	E_MA_EVENT.STOP_TRACK:
		RefStat.sm.sEventDesc := 'CMD STOP_TRACK';
		RETURN;
		
	E_MA_EVENT.PRESETDONE:
		RefStat.sm.sEventDesc := 'TRACKING';
		RETURN;
		
	E_MA_EVENT.TRACKEXIT:
		RefStat.sm.sEventDesc := 'TRACKING -> PRESETTING';
		RETURN;
		
	E_MA_EVENT.HWOK:
		RefStat.sm.sEventDesc := 'SIG HWOK';
		RETURN;

	E_MA_EVENT.ERRHW:
		RefStat.sm.sEventDesc := 'INT ERRHW';
		RETURN;
	
END_CASE 

(* INTERNAL ERROR *)
RefStat.sm.sEventDesc := 'UNKNOWN EVENT';
END_METHOD

// Set the state and substate of the device
METHOD SetState : BOOL
VAR_INPUT
	in_nState:		INT;
	in_nSubstate:	INT;
END_VAR

(* 
	Update State Machine active state configuration.
*)

IF in_nState <> E_MA_STATE.NONE THEN
	RefStat.sm.nState	:= in_nState;
END_IF
IF in_nSubstate <> E_MA_SUBSTATE.NONE THEN
	RefStat.sm.nSubstate	:= in_nSubstate;
END_IF

(* Update active state configuration description *)

IF in_nState = E_MA_STATE.NOTOP THEN
	RefStat.sm.sState	:= 'NOT OP';
ELSIF in_nState = E_MA_STATE.OP THEN
	RefStat.sm.sState	:= 'OPERATIONAL';
END_IF

IF in_nSubstate = E_MA_SUBSTATE.NOTOP_NOTREADY THEN
	RefStat.sm.sSubstate	:= 'NOT READY';
ELSIF in_nSubstate = E_MA_SUBSTATE.NOTOP_INITIALISING THEN
	RefStat.sm.sSubstate	:= 'INITIALISING';
ELSIF in_nSubstate = E_MA_SUBSTATE.NOTOP_READY THEN
	RefStat.sm.sSubstate	:= 'READY';
ELSIF in_nSubstate = E_MA_SUBSTATE.NOTOP_ERROR THEN
	RefStat.sm.sSubstate	:= 'ERROR';
ELSIF in_nSubstate = E_MA_SUBSTATE.OP_DISABLING THEN
	RefStat.sm.sSubstate	:= 'DISABLING';
ELSIF in_nSubstate = E_MA_SUBSTATE.OP_MOVING THEN
	RefStat.sm.sSubstate	:= 'MOVING';
ELSIF in_nSubstate = E_MA_SUBSTATE.OP_STANDSTILL THEN
	RefStat.sm.sSubstate	:= 'STANDSTILL';
ELSIF in_nSubstate = E_MA_SUBSTATE.OP_TRACKING THEN
	RefStat.sm.sSubstate	:= 'TRACKING';
ELSIF in_nSubstate = E_MA_SUBSTATE.OP_PRESETTING THEN
	RefStat.sm.sSubstate	:= 'PRESETTING';
ELSIF in_nSubstate = E_MA_SUBSTATE.OP_STOPPING THEN
	RefStat.sm.sSubstate	:= 'STOPPING';
ELSIF in_nSubstate = E_MA_SUBSTATE.OP_ERROR THEN
	RefStat.sm.sSubstate	:= 'ERROR';
ELSE
	RefStat.sm.sSubstate	:= '';
END_IF
END_METHOD

METHOD User_ComputeNextPos : BOOL
VAR_INPUT
END_VAR
VAR
	i:	int;
END_VAR
// TODOUSER: Calculate next position for each axes based on the current mode.
IF RefStat.nMode = MA_MODE_ENG THEN
	FOR i := 1 TO nNumAxes DO
		;
	END_FOR
END_IF
END_METHOD

// Method for hard-coding of configuration parameters by the User.
METHOD User_Configure : BOOL
VAR_INPUT
END_VAR
VAR
	i:	INT;
END_VAR
//
// TODOUSER: Configure anything that is different from default configuration or
//           that has to take all motors into account.
//

//
// This is mandatory.
//
// Set the global timeouts to the longest ones. 
FOR i := 1 TO nNumAxes DO
	IF ptrMotorCfg[i]^.nTimeoutInit > RefCfg.tout.initTime THEN
		RefCfg.tout.initTime  := ptrMotorCfg[i]^.nTimeoutInit;
	END_IF
	IF ptrMotorCfg[i]^.nTimeoutMove > RefCfg.tout.moveTime THEN
		RefCfg.tout.moveTime  := ptrMotorCfg[i]^.nTimeoutMove;
	END_IF
END_FOR

//
// TODOUSER: Any other configuration
//
END_METHOD

// User Method executed on each cycle before processing events and states.
METHOD User_GetParams : BOOL
VAR_INPUT
END_VAR
VAR
	i:	INT;
END_VAR
//
// TODOUSER: Set anything that should be set on every cycle, if any.
//

// Example: Any settings that are mode dependant.
CASE RefCtrl.nMode OF
			MA_MODE_ENG:
			    ; 
END_CASE
END_METHOD

// User Method executed on each cycle after processing events and states.
METHOD User_SetParams : BOOL
VAR_INPUT
END_VAR
VAR
	i:		INT;
END_VAR
//
// Mandatory
//
// Set maximum positioning error
RefStat.lrPosError	:= M_GetMaxPosError();


// TODO Add code for handling individual axes, if any.
FOR i := 1 TO nNumAxes DO
	;
END_FOR
END_METHOD

END_FUNCTION_BLOCK

// POUs/MultiAxis/FB_MA_DROT
FUNCTION_BLOCK FB_MA_DROT EXTENDS FB_TRK_BASE
VAR_INPUT
	{attribute 'OPC.UA.DA' := '0'}
	sMotorName:			STRING	:= 'Motor';	(* Default Motor name *)
	{attribute 'OPC.UA.DA' := '0'}
	nNOVRAM_DevId:	UDINT	:= 0;		(* NOVRAM device ID - normally 4 *)
	{attribute 'OPC.UA.DA' := '0'}
	nNOVRAM_Offset:	UDINT	:= 0;		(* NOVRAM offset where motor configuration is stored *)
END_VAR
VAR_OUTPUT
END_VAR
VAR

	
	{attribute 'OPC.UA.DA' := '1'}
	cfg:				T_DROT_CFG;
	{attribute 'OPC.UA.DA' := '1'}
	ctrl:				T_DROT_CTRL;
	{attribute 'OPC.UA.DA' := '1'}
	stat:				T_DROT_STAT;
	
	{attribute 'OPC.UA.DA':='1'}
	motor:              FB_MOTOR;
	
END_VAR


// A MUST !!! Set references to real structures
RefCfg		REF=cfg;
RefCtrl		REF=ctrl;
RefStat		REF=stat;
TrkStat		REF=stat;
TrkCfg      REF=cfg;
TrkCtrl     REF=ctrl;

motor(sName := sMotorName,	nNOVRAM_DevId := nNOVRAM_DevId, nNOVRAM_Offset := nNOVRAM_Offset);
SUPER^(nNumAxes:=1, pMotor1:=ADR(motor));

METHOD M_LogCommand : BOOL
VAR
	cmd:	INT;
	mode:	int;
END_VAR
cmd		:= RefCtrl.nCommand;
mode	:= ctrl.nMode;

// Log DROT command.
// Set motor logging to FALSE when tracking,
// in order to reduce flooding of logs.
IF cmd = E_MA_COMMAND.RESET THEN
	pMotor1^.RPC_SetLog(TRUE);
	M_SetStatus('Resetting DROT device...');		
	M_LogEventGeneral('Resetting DROT device...');
ELSIF cmd = E_MA_COMMAND.ENABLE THEN
	pMotor1^.RPC_SetLog(TRUE);
	M_SetStatus('');		
	M_LogEventGeneral('Enabling DROT device...');
ELSIF cmd = E_MA_COMMAND.INIT THEN
	pMotor1^.RPC_SetLog(TRUE);
	M_SetStatus('Initialising DROT device...');		
	M_LogEventGeneral('Initialising DROT device...');
ELSIF cmd = E_MA_COMMAND.START_TRACK THEN
	pMotor1^.RPC_SetLog(FALSE);
	IF mode= E_DROT_MODE.ELEV THEN
		M_SetStatus('Tracking in ELEV mode');
		M_LogEventGeneral('Setting DROT device to ELEVATION mode...');
	ELSIF mode= E_DROT_MODE.SKY THEN
		M_SetStatus('Tracking in SKY mode');
		M_LogEventGeneral('Setting DROT device to SKY mode...');
	ELSIF mode= E_DROT_MODE.USER THEN
		M_SetStatus('Tracking in USER mode');
		M_LogEventGeneral('Setting DROT device to USER mode...');
	END_IF
ELSIF cmd = E_MA_COMMAND.DISABLE THEN
	M_SetStatus('');		
	M_LogEventGeneral('Disabling DROT device...');
ELSIF cmd = E_MA_COMMAND.STOP THEN
	pMotor1^.RPC_SetLog(TRUE);
	M_LogEventGeneral('Stopping DROT device...');
ELSIF cmd = E_MA_COMMAND.STOP_TRACK THEN
	pMotor1^.RPC_SetLog(TRUE);
	IF mode= E_DROT_MODE.ENG THEN
		M_SetStatus('Moving to Engineering position ...');		
		M_LogEventGeneral('Setting DROT device to ENGINEERING mode...');
	ELSIF mode= E_DROT_MODE.STAT THEN
		M_SetStatus('Moving to STAT position ...');		
		M_LogEventGeneral('Setting DROT device to STAT mode...');
	END_IF
END_IF
END_METHOD

{attribute 'TcRpcEnable':='1'}
METHOD RPC_Disable : INT
VAR_INPUT
END_VAR

// It does all the verifications for the MOTOR device before
// triggering the Init event.

// RPC calls are not allowed in Local mode.
IF ptrMotorStat[1]^.bLocal THEN
	RPC_Disable	:= M_SetRpcStatus(E_MA_RPC_ERROR.LOCAL);
	RETURN;
END_IF

// Disable command is accepted only if device is in OP state.
IF ptrMotorStat[1]^.nState <> E_MOTOR_STATE.OP THEN
	RPC_Disable	:= M_SetRpcStatus(E_MA_RPC_ERROR.NOT_OP);
	RETURN;
ELSE
	// Set disable command
	RefCtrl.nCommand := E_MA_COMMAND.DISABLE;
	RefCtrl.bExecute := TRUE;
	
	// Call was successful
	RPC_Disable	:= M_SetRpcStatus(E_MA_RPC_ERROR.OK);
END_IF
END_METHOD

{attribute 'TcRpcEnable':='1'}
METHOD RPC_Enable : INT
VAR_INPUT
END_VAR

// It does all the verifications for the MOTOR device before
// triggering the Init event.


// RPC calls are not allowed in Local mode.
IF ptrMotorStat[1]^.bLocal THEN
	RPC_Enable	:= M_SetRpcStatus(E_MA_RPC_ERROR.LOCAL);
	RETURN;
END_IF

// Enable command is accepted only if device is in NOTOP_READY.
IF	ptrMotorStat[1]^.nSubstate <> E_MOTOR_SUBSTATE.NOTOP_READY		THEN
	RPC_Enable	:= M_SetRpcStatus(E_MA_RPC_ERROR.NOT_NOTOP_READY);
	RETURN;
ELSE
	// Set enable command
	RefCtrl.nCommand := E_MA_COMMAND.ENABLE;
	RefCtrl.bExecute := TRUE;
	
	// Call was successful
	RPC_Enable	:= M_SetRpcStatus(E_MA_RPC_ERROR.OK);
END_IF
END_METHOD

{attribute 'TcRpcEnable':='1'}
METHOD RPC_Init : INT
VAR_INPUT
END_VAR

VAR
END_VAR
M_LogEventGeneral('Initialising DROT motor...');

RPC_Init	:= SUPER^.RPC_Init();
END_METHOD

{attribute 'TcRpcEnable':='1'}
METHOD RPC_MoveAbs : INT
VAR_INPUT
	in_lrPos:	LREAL;
	in_lrVel:	LREAL;
END_VAR
// RPC calls are not allowed in Local mode.
IF motor.stat.bLocal THEN
	RPC_MoveAbs	:= M_SetRpcStatus(E_MA_RPC_ERROR.LOCAL);
	RETURN;
// Move Absolute command is accepted only in OP state.
ELSIF	motor.stat.nState <> E_MOTOR_STATE.OP	THEN
	RPC_MoveAbs	:= M_SetRpcStatus(E_MA_RPC_ERROR.NOT_OP);
	RETURN;
ELSIF	stat.sm.nState <> E_MA_STATE.OP	THEN
	RPC_MoveAbs	:= M_SetRpcStatus(E_MA_RPC_ERROR.NOT_OP);
	RETURN;
// Set velocity cannot be <=0.0.
ELSIF	in_lrVel <= 0.0	THEN
	RPC_MoveAbs	:= M_SetRpcStatus(E_MOTOR_RPC_ERROR.VEL_NEG);
	RETURN;
// Set velocity cannot be greater than MAX Velocity.
ELSIF	in_lrVel > motor.stat.axis.lrMaxVelocity	THEN
	RPC_MoveAbs	:= M_SetRpcStatus(E_MOTOR_RPC_ERROR.VEL_MAX);
	RETURN;
END_IF


SetState(E_MA_STATE.OP, E_MA_SUBSTATE.OP_MOVING);
// Set command
ctrl.nCommand 		:= E_MA_COMMAND.MA_MOVE;
ctrl.nMode          := E_DROT_MODE.ENG;
ctrl.lrTargetPos    := in_lrPos;
ctrl.lrTargetVel    := in_lrVel;
ctrl.bExecute 		:= TRUE;

// Call was successful
RPC_MoveAbs	:= M_SetRpcStatus(E_MA_RPC_ERROR.OK);
END_METHOD

{attribute 'TcRpcEnable':='1'}
METHOD RPC_MoveAngle : INT
VAR_INPUT
	in_lrAngle:	LREAL;
END_VAR

// RPC calls are not allowed in Local mode.
IF motor.stat.bLocal THEN
	RPC_MoveAngle	:= M_SetRpcStatus(E_MA_RPC_ERROR.LOCAL);
	RETURN;
// Move Absolute command is accepted only in OP state.
ELSIF	motor.stat.nState <> E_MOTOR_STATE.OP	THEN
	RPC_MoveAngle	:= M_SetRpcStatus(E_MA_RPC_ERROR.NOT_OP);
	RETURN;
ELSIF	stat.sm.nState <> E_MA_STATE.OP	THEN
	RPC_MoveAngle	:= M_SetRpcStatus(E_MA_RPC_ERROR.NOT_OP);
	RETURN;
END_IF


SetState(E_MA_STATE.OP, E_MA_SUBSTATE.OP_MOVING);
// Set command
ctrl.lrPosang 	:= in_lrAngle;
ctrl.nMode		:= E_DROT_MODE.STAT;
ctrl.nCommand	:= E_MA_COMMAND.STOP_TRACK;
ctrl.bExecute	:= TRUE;

// Call was successful
RPC_MoveAngle	:= M_SetRpcStatus(E_MA_RPC_ERROR.OK);
END_METHOD

{attribute 'TcRpcEnable':='1'}
METHOD RPC_MoveRel : INT
VAR_INPUT
	in_lrPos:	LREAL;
	in_lrVel:	LREAL;
END_VAR
// RPC calls are not allowed in Local mode.
IF motor.stat.bLocal THEN
	RPC_MoveRel	:= M_SetRpcStatus(E_MA_RPC_ERROR.LOCAL);
	RETURN;
// Move Absolute command is accepted only in OP state.
ELSIF	motor.stat.nState <> E_MOTOR_STATE.OP	THEN
	RPC_MoveRel	:= M_SetRpcStatus(E_MA_RPC_ERROR.NOT_OP);
	RETURN;
ELSIF	stat.sm.nState <> E_MA_STATE.OP	THEN
	RPC_MoveRel	:= M_SetRpcStatus(E_MA_RPC_ERROR.NOT_OP);
	RETURN;
// Set velocity cannot be <=0.0.
ELSIF	in_lrVel <= 0.0	THEN
	RPC_MoveRel	:= M_SetRpcStatus(E_MOTOR_RPC_ERROR.VEL_NEG);
	RETURN;
// Set velocity cannot be greater than MAX Velocity.
ELSIF	in_lrVel > motor.stat.axis.lrMaxVelocity	THEN
	RPC_MoveRel	:= M_SetRpcStatus(E_MOTOR_RPC_ERROR.VEL_MAX);
	RETURN;
END_IF


SetState(E_MA_STATE.OP, E_MA_SUBSTATE.OP_MOVING);
// Set command
ctrl.nCommand 		:= E_MA_COMMAND.MA_MOVE;
ctrl.nMode          := E_DROT_MODE.ENG;
ctrl.lrTargetPos    := motor.stat.lrPosActual + in_lrPos;
ctrl.lrTargetVel    := in_lrVel;
ctrl.bExecute 		:= TRUE;

// Call was successful
RPC_MoveRel	:= M_SetRpcStatus(E_MA_RPC_ERROR.OK);
END_METHOD

{attribute 'TcRpcEnable':='1'}
METHOD RPC_MoveVel : INT
VAR_INPUT
	in_lrVel:	LREAL;
END_VAR
VAR
	dir:	DINT;
END_VAR
IF	stat.sm.nState <> E_MA_STATE.OP	THEN
	RPC_MoveVel	:= M_SetRpcStatus(E_MA_RPC_ERROR.NOT_OP);
	RETURN;
ELSIF	in_lrVel = 0.0	THEN
// Set velocity cannot be 0.0.
	RPC_MoveVel	:= M_SetRpcStatus(E_MOTOR_RPC_ERROR.VEL_ZERO);
	RETURN;
END_IF

// Check velocity against Vel_max.
// Note: Negative velocity is accepted.
// Check if Velocity is too high.
IF ABS(in_lrVel) > ptrMotorStat[1]^.axis.lrMaxVelocity THEN
	RPC_MoveVel	:= M_SetRpcStatus(E_MOTOR_RPC_ERROR.VEL_MAX);
	RETURN;
END_IF


// Update State and Status
SetState(E_MA_STATE.OP, E_MA_SUBSTATE.OP_MOVING);
M_SetStatus('Moving in Velocity mode...');
ctrl.nMode	:= E_ADC_MODE.ENG;

// Set the direction of movement.
IF in_lrVel > 0.0	THEN
	dir	:= MC_Positive_Direction;
ELSE
	dir	:= MC_Negative_Direction;
END_IF

// This will command all the motors and restart the timer.
ActionMoveVelExecute(vel:=ABS(in_lrVel), dir:=dir);

// Call was successful
RPC_MoveVel	:= M_SetRpcStatus(E_MA_RPC_ERROR.OK);
END_METHOD

{attribute 'TcRpcEnable':='1'}
METHOD RPC_Reset : INT
VAR_INPUT
END_VAR

// RPC calls are not allowed in Local mode.
IF ptrMotorStat[1]^.bLocal THEN
	RPC_Reset	:= M_SetRpcStatus(E_MA_RPC_ERROR.LOCAL);
	RETURN;
END_IF

ctrl.nCommand := E_MA_COMMAND.RESET;
ctrl.bExecute := TRUE;

// Call was successful
RPC_Reset	:= M_SetRpcStatus(E_MA_RPC_ERROR.OK);
END_METHOD

{attribute 'TcRpcEnable':='1'}
METHOD RPC_StartTrack : INT
VAR_INPUT
	in_mode:	 INT := 2;
	in_angle:    LREAL := 0.0;
END_VAR

// RPC calls are not allowed in Local mode.
IF ptrMotorStat[1]^.bLocal THEN
	RPC_StartTrack	:= M_SetRpcStatus(E_MA_RPC_ERROR.LOCAL);
	RETURN;
// Move Absolute command is accepted only in OP state.
ELSIF	ptrMotorStat[1]^.nState <> E_MOTOR_STATE.OP	THEN
	RPC_StartTrack	:= M_SetRpcStatus(E_MA_RPC_ERROR.NOT_OP);
	RETURN;
END_IF

// Set command
ctrl.lrPosang := in_angle;
ctrl.nMode:= in_mode;
ctrl.nCommand:=E_MA_COMMAND.START_TRACK;
ctrl.bExecute:=(TRUE);

// Call was successful
RPC_StartTrack	:= M_SetRpcStatus(E_MA_RPC_ERROR.OK);
END_METHOD

{attribute 'TcRpcEnable':='1'}
METHOD RPC_Stop : INT
VAR_INPUT
END_VAR

// RPC calls are not allowed in Local mode.
IF ptrMotorStat[1]^.bLocal THEN
	RPC_Stop	:= M_SetRpcStatus(E_MA_RPC_ERROR.LOCAL);
	RETURN;
END_IF

ctrl.nCommand := E_MA_COMMAND.STOP;
ctrl.bExecute := TRUE;

RPC_Stop	:= M_SetRpcStatus(E_MA_RPC_ERROR.OK);
END_METHOD

{attribute 'TcRpcEnable':='1'}
METHOD RPC_StopTrack : INT
VAR_INPUT
END_VAR

IF (RefStat.nMode >= E_DROT_MODE.SKY) THEN
	// RPC calls are not allowed in Local mode.
	IF ptrMotorStat[1]^.bLocal THEN
		RPC_StopTrack	:= M_SetRpcStatus(E_MA_RPC_ERROR.LOCAL);
		RETURN;
	END_IF

	RefCtrl.nMode           :=  E_DROT_MODE.STAT;
	// Set command
	RefCtrl.nCommand 		:= E_MA_COMMAND.STOP_TRACK;
	RefCtrl.bExecute 		:= TRUE;
END_IF

// Call was successful
RPC_StopTrack	:= M_SetRpcStatus(E_MA_RPC_ERROR.OK);
END_METHOD

METHOD User_ComputeNextPos : BOOL
VAR_INPUT
END_VAR
VAR
	fieldRotation: LREAL;
	modeAngle:     LREAL;
	pos:           LREAL := 0.0 ;
	posang:        LREAL;
END_VAR
// Handle various derotator modes
CASE RefCtrl.nMode OF
			E_DROT_MODE.STAT:
			    pos := cfg.lrStatRef + cfg.nDirSign * (ctrl.lrPosang)/2.0;
				stat.lrAngleOnSky := 0.0;
				stat.lrModeAngle := pos;
				ptrMotorCtrl[1]^.lrVelocity := ptrMotorCfg[1]^.lrDefaultVelocity;
			E_DROT_MODE.SKY:
				fieldRotation := stat.data.pa_deg - cfg.nFocusSign * stat.data.alt_deg;
				pos := cfg.lrSkyRef + cfg.nDirSign * (ctrl.lrPosang - fieldRotation)/2;
				stat.lrAngleOnSky := ctrl.lrPosang;
				stat.lrModeAngle := stat.lrAngleOnSky;
				ptrMotorCtrl[1]^.lrVelocity := ptrMotorCfg[1]^.lrDefaultVelocity;
			E_DROT_MODE.ELEV:
				pos := cfg.lrElevRef + (cfg.nFocusSign * cfg.nDirSign * stat.data.alt_deg) /2.0;
				stat.lrAngleOnSky := stat.data.pa_deg;
				stat.lrModeAngle := stat.lrAngleOnSky;
				ptrMotorCtrl[1]^.lrVelocity := ptrMotorCfg[1]^.lrDefaultVelocity;
			E_DROT_MODE.USER:
				//modeAngle := (parUser[1] * ctrl.lrPosang +
				//	          parUser[2] * i_trk_data.alt_deg +
				//			  parUser[3] * i_trk_data.pa_deg );
				//pos := cfg.lrUserRef + cfg.nDirSign * modeAngle;
				//stat.lrAngleOnSky := 0.0;
				//stat.lrModeAngle  := modeAngle;
			E_DROT_MODE.ENG:
				pos := ctrl.lrTargetPos;
		        ptrMotorCtrl[1]^.lrVelocity := ctrl.lrTargetVel;		
		        M_SetStatus('Moving to Engineering position ...');
END_CASE

// assign new TARGET position
ptrMotorCtrl[1]^.lrPosition := pos;
stat.lrPos := pos;	// Used in the DROT GUI as 'Target'
END_METHOD

// Method for hard-coding of configuration parameters by the User.
METHOD User_Configure : BOOL
VAR_INPUT
END_VAR
VAR
	i:	INT;
END_VAR
SUPER^.User_Configure();	// Mandatory!

//
// TODOUSER: Configure anything that is different from default configuration.
//
// Examples:
//

//
// Individual Motor configuration
ptrMotorCfg[1]^.nAxisType	        := E_MOTOR_AXIS_TYPE.CIRCULAR_OPTIMISED;
ptrMotorCfg[1]^.lrDefaultVelocity	:= 3.0;	// Set default velocity to 10 deg/sec


// Multi-axis system configuration
ctrl.lrPosang	    :=  0.0;	// Position angle for OFF mode, i.e. HOME position
ctrl.lrTargetPos	:=  0.0;	
ctrl.lrTargetVel	:= 3.0;	// Velocity for ENG mode
END_METHOD

// User Method executed on each cycle before processing events and states.
METHOD User_GetParams : BOOL
VAR_INPUT
END_VAR
VAR
	i:	INT;
END_VAR


SUPER^.User_GetParams();
END_METHOD

// User Method executed on each cycle after processing events and states.
METHOD User_SetParams : BOOL
VAR_INPUT
END_VAR
VAR
	i:		INT;
END_VAR
//
// Mandatory
//
SUPER^.User_SetParams();

// Set maximum positioning error
stat.lrPosError		:= M_GetMaxPosError();

// Check if we are tracking or still presetting.
// Tracking is OK if the positioning error is less than the threshold (bTrackingOK).
// Once device is tracking, it should go back to presetting if the error is greater
// than twice the threshold  (bTrackingBAD).
IF	ctrl.nMode = E_DROT_MODE.ELEV OR  
	ctrl.nMode = E_DROT_MODE.SKY  OR  
	ctrl.nMode = E_DROT_MODE.USER	THEN
	stat.bTrackingOK	:= SEL (stat.lrPosError <= cfg.lrTrkThreshold, FALSE, TRUE);
	stat.bTrackingBAD	:= SEL (stat.lrPosError > 2.0 * cfg.lrTrkThreshold, FALSE, TRUE);
ELSE
	stat.bTrackingOK	:= FALSE;
	stat.bTrackingBAD	:= FALSE;
END_IF
END_METHOD

END_FUNCTION_BLOCK

// VISUs/Motor/GUI_Motor001_Cfg
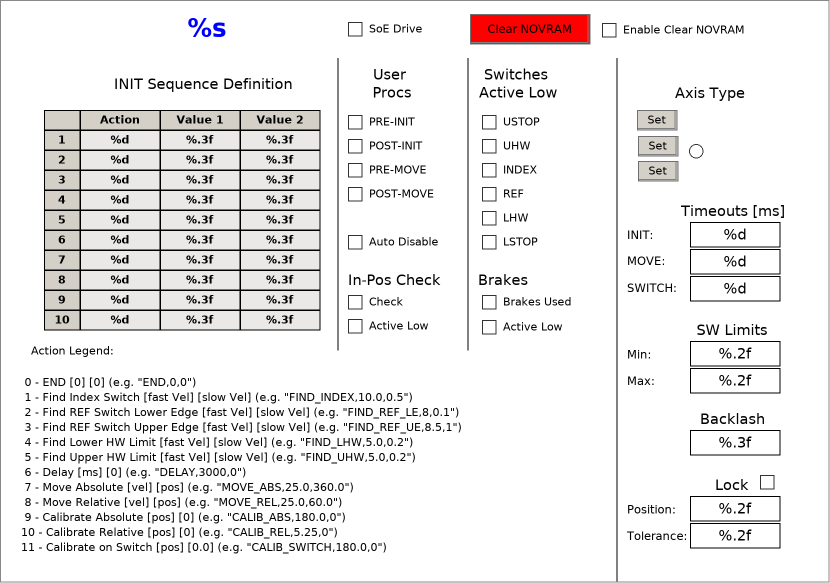
VISUALIZATION GUI_Motor001_Cfg  // 830x583
    Frame (0,0 828x581)
        shows GUI_TEMPLATE_MOTOR_CONFIG(m_Instance := MAIN.Motor001)
END_VISUALIZATION

// VISUs/Motor/GUI_Motor001_Ctrl
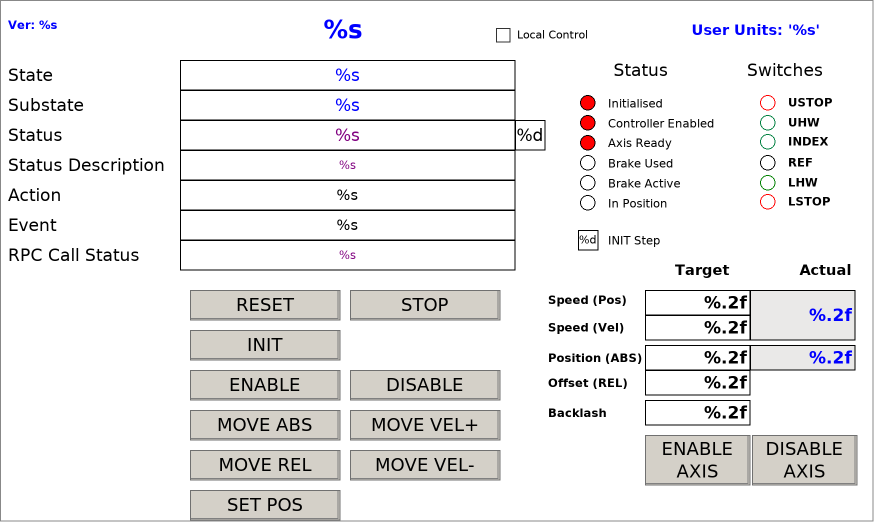
VISUALIZATION GUI_Motor001_Ctrl  // 874x522
    Frame (0,0 872x520)
        shows GUI_TEMPLATE_MOTOR_CONTROL(m_Instance := MAIN.Motor001)
END_VISUALIZATION

// VISUs/Motor/GUI_Motor002_Cfg
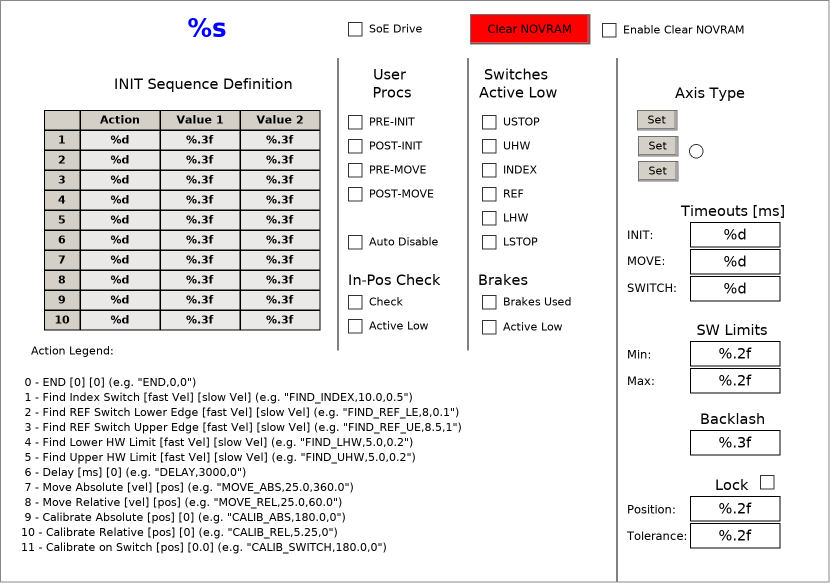
VISUALIZATION GUI_Motor002_Cfg  // 830x583
    Frame (0,0 828x581)
        shows GUI_TEMPLATE_MOTOR_CONFIG(m_Instance := MAIN.Motor002)
END_VISUALIZATION

// VISUs/Motor/GUI_Motor002_Ctrl
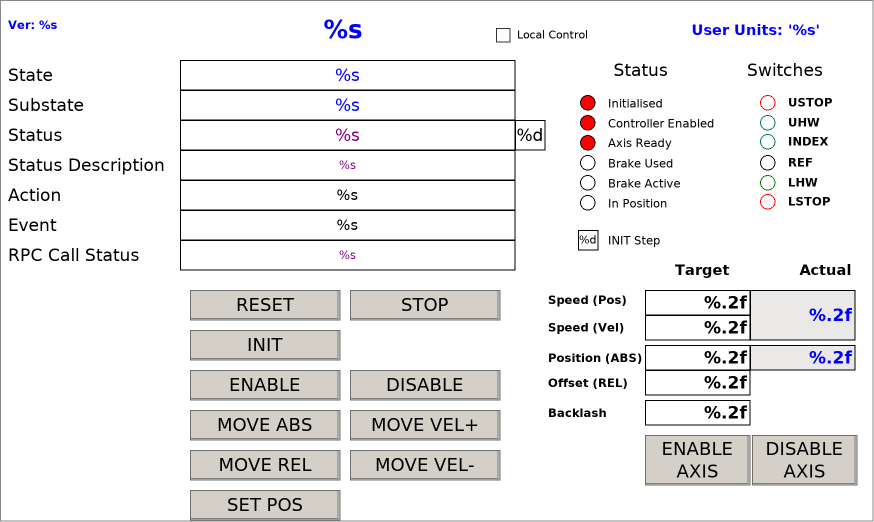
VISUALIZATION GUI_Motor002_Ctrl  // 874x522
    Frame (0,0 872x520)
        shows GUI_TEMPLATE_MOTOR_CONTROL(m_Instance := MAIN.Motor002)
END_VISUALIZATION

// VISUs/Templates/GUI_TEMPLATE_CCS_SIM
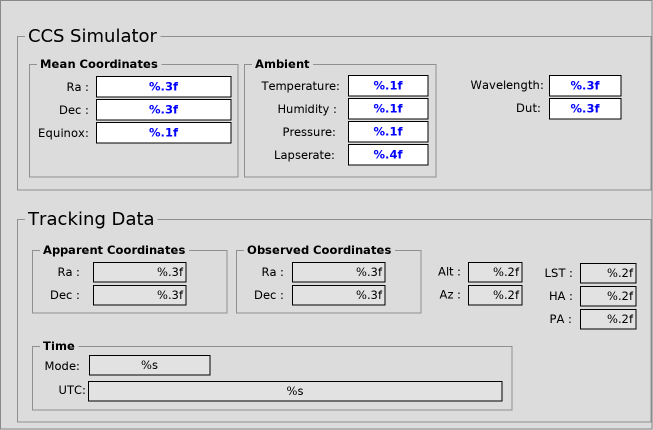
VISUALIZATION GUI_TEMPLATE_CCS_SIM  // 653x430
VAR_INPUT
	m_DeviceName : STRING;
END_VAR
VAR_IN_OUT
	m_Instance : FB_CCS_SIM;
END_VAR
    GroupBox (17,28 634x162), "CCS Simulator"
        GroupBox (12,28 209x121), "Mean Coordinates"
            Label (23,21 40x20), "Ra :"
            Label (23,44 40x20), "Dec :"
            Rectangle (67,20 135x21), "%.3f", tooltip "Mean Right Ascension [hhmmss]", text variable: m_Instance.ctrl.meanCoordinates.alpha
                OnMouseDown: write the text variable via Edit
            Rectangle (67,43 135x21), "%.3f", tooltip "Mean Declination [ddmmss]", text variable: m_Instance.ctrl.meanCoordinates.delta
                OnMouseDown: write the text variable via Edit
            Rectangle (67,66 135x21), "%.1f", tooltip "Equinox", text variable: m_Instance.ctrl.meanCoordinates.equinox
                OnMouseDown: write the text variable via Edit
            Label (3,67 60x20), "Equinox:"
        GroupBox (227,28 192x121), "Ambient"
            Label (7,20 92x20), "Temperature:"
            Label (17,43 79x20), "Humidity :"
            Rectangle (104,19 80x21), "%.1f", tooltip "Temperature [degC]", text variable: m_Instance.ctrl.environment.temperature
                OnMouseDown: write the text variable via Edit
            Rectangle (104,42 80x21), "%.1f", tooltip "Humidity [%]", text variable: m_Instance.ctrl.environment.humidity
                OnMouseDown: write the text variable via Edit
            Rectangle (104,65 80x21), "%.1f", tooltip "Pressure [mbar]", text variable: m_Instance.ctrl.environment.pressure
                OnMouseDown: write the text variable via Edit
            Label (25,66 70x20), "Pressure:"
            Label (24,89 70x20), "Lapserate:"
            Rectangle (104,88 80x21), "%.4f", tooltip "Lapse Rate", text variable: m_Instance.ctrl.environment.lapserate
                OnMouseDown: write the text variable via Edit
        Rectangle (532,47 72x21), "%.3f", text variable: m_Instance.ctrl.wavelength
            OnMouseDown: write the text variable via Edit
        Rectangle (532,70 72x21), "%.3f", text variable: m_Instance.ctrl.dut
            OnMouseDown: write the text variable via Edit
        Label (481,70 46x20), "Dut:"
    GroupBox (17,211 634x211), "Tracking Data"
        GroupBox (15,31 195x71), "Apparent Coordinates"
            Label (11,20 40x20), "Ra :"
            Label (11,43 40x20), "Dec :"
            Label (8,70 60x20)
            Rectangle (61,43 93x20), "%.3f", tooltip "Apparent Declination [ddmmss]", text variable: m_Instance.stat.apparent.delta
            Rectangle (61,20 93x20), "%.3f", tooltip "Apparent Right Ascension [hhmmss]", text variable: m_Instance.stat.apparent.alpha
        Rectangle (563,98 56x20), "%.2f", tooltip "Parallactic Angle [deg]", text variable: m_Instance.stat.data.pa_deg
        Label (508,98 50x20), "PA :"
        Label (410,51 37x19), "Alt :"
        Label (412,74 35x19), "Az :"
        GroupBox (219,31 185x71), "Observed Coordinates"
            Label (11,20 40x20), "Ra :"
            Label (11,43 40x20), "Dec :"
            Label (8,70 60x20)
            Rectangle (56,20 93x20), "%.3f", tooltip "Observed Right Ascension [hhmmss]", text variable: m_Instance.stat.observed.alpha
            Rectangle (56,43 93x20), "%.3f", tooltip "Observed Declination [ddmmss]", text variable: m_Instance.stat.observed.delta
        Rectangle (451,74 54x20), "%.2f", tooltip "TEL Azimuth [deg]", text variable: m_Instance.stat.data.az_deg
        Rectangle (451,51 54x20), "%.2f", tooltip "TEL Altitude [deg]", text variable: m_Instance.stat.data.alt_deg
        GroupBox (15,127 480x72), "Time"
            Label (11,18 40x20), "Mode:"
            Label (11,42 46x20), "UTC:"
            Label (8,70 60x20)
            Rectangle (57,17 121x20), "%s", tooltip "Time mode [UTC, Local or Simulation]", text variable: m_Instance.stat.sTimeMode
            Rectangle (56,43 414x20), "%s", tooltip "Actual time", text variable: m_Instance.stat.sDcTime
    Label (464,75 83x20), "Wavelength:"
    Label (526,263 50x20), "LST :"
    Label (526,286 50x20), "HA :"
    Rectangle (580,286 56x20), "%.2f", tooltip "Hour Angle [deg]", text variable: m_Instance.stat.data.ha
    Rectangle (580,263 56x20), "%.2f", tooltip "Local Sidereal Time [h]", text variable: m_Instance.stat.data.lst
END_VISUALIZATION

// VISUs/Templates/GUI_TEMPLATE_MA_ADC
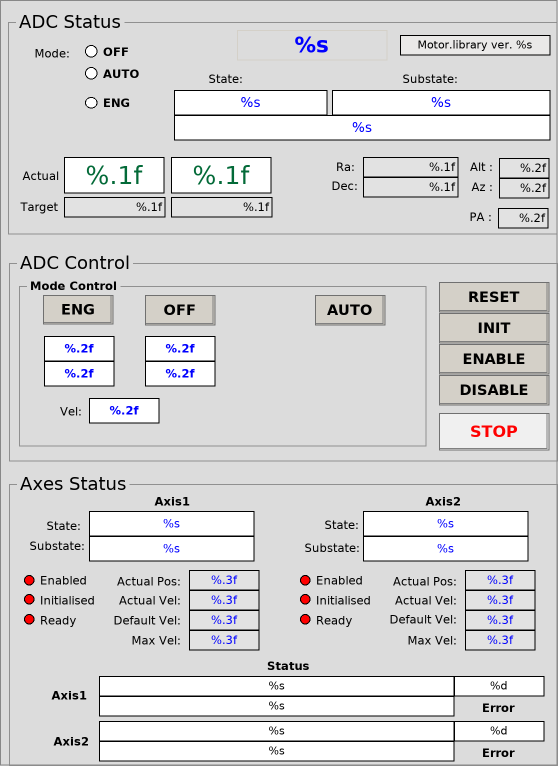
VISUALIZATION GUI_TEMPLATE_MA_ADC  // 558x766
VAR_INPUT
	m_DeviceName : STRING;
END_VAR
VAR_IN_OUT
	m_Instance : FB_MA_ADC;
END_VAR
    GroupBox (9,255 549x206), "ADC Control"
        Button (430,158 110x37), "STOP"
            OnMouseClick: execute { m_Instance.ctrl.nCommand:= E_MA_COMMAND.STOP; m_Instance.ctrl.bExecute:=(TRUE); }
        GroupBox (10,23 407x168), "Mode Control"
            Button (296,17 70x30), "AUTO", tooltip "Tracking mode (2)"
                OnMouseClick: execute {
                    m_Instance.ctrl.nMode:= E_ADC_MODE.AUTO;
                    m_Instance.ctrl.nCommand:=E_MA_COMMAND.START_TRACK;
                    m_Instance.ctrl.bExecute:=(TRUE);
                }
            Rectangle (70,120 70x25), "%.2f", tooltip "Velocity for Engineering Mode [deg/sec]", text variable: m_Instance.ctrl.lrTargetVel
                OnMouseDown: write the text variable via Edit
            Button (126,17 70x30), "OFF", tooltip "OFF (HOME) mode (1)"
                OnMouseClick: execute {
                    m_Instance.ctrl.nMode:=E_ADC_MODE.OFF;
                    m_Instance.ctrl.nCommand:= E_MA_COMMAND.STOP_TRACK;
                    m_Instance.ctrl.bExecute:=(TRUE);
                }
            Label (36,121 30x25), "Vel:"
            Rectangle (126,58 70x25), "%.2f", tooltip "ADC1 OFF Position angle [deg]", text variable: m_Instance.ctrl.lrPosang[1]
                OnMouseDown: write the text variable via Edit
            Rectangle (126,83 70x25), "%.2f", tooltip "ADC2 OFF position angle [deg]", text variable: m_Instance.ctrl.lrPosang[2]
                OnMouseDown: write the text variable via Edit
            Button (24,17 70x29), "ENG", tooltip "ENG mode (0)"
                OnMouseClick: execute {
                    m_Instance.ctrl.nMode:=E_ADC_MODE.ENG;
                    m_Instance.ctrl.nCommand:= E_MA_COMMAND.STOP_TRACK;
                    m_Instance.ctrl.bExecute:=(TRUE);
                }
            Rectangle (25,58 70x25), "%.2f", tooltip "ADC1 ENG Position angle [deg]", text variable: m_Instance.ctrl.lrTargetPos[1]
                OnMouseDown: write the text variable via Edit
        Button (430,120 110x30), "DISABLE"
            OnMouseClick: execute { m_Instance.ctrl.nCommand:= E_MA_COMMAND.DISABLE; m_Instance.ctrl.bExecute:=(TRUE); }
        Button (430,27 110x30), "RESET"
            OnMouseClick: execute { m_Instance.ctrl.nCommand:= E_MA_COMMAND.RESET; m_Instance.ctrl.bExecute:=(TRUE); }
        Button (430,89 110x30), "ENABLE"
            OnMouseClick: execute { m_Instance.ctrl.nCommand:= E_MA_COMMAND.ENABLE; m_Instance.ctrl.bExecute:=(TRUE); }
        Button (430,58 110x30), "INIT"
            OnMouseClick: execute { m_Instance.ctrl.nCommand:= E_MA_COMMAND.INIT; m_Instance.ctrl.bExecute:=(TRUE); }
    GroupBox (9,476 549x290), "Axes Status"
        Label (98,93 77x25), "Actual Pos:"
        Rectangle (180,94 70x20), "%.3f", tooltip "[deg]", text variable: m_Instance.pMotor1^.stat.lrPosActual
        Rectangle (180,114 70x20), "%.3f", tooltip "[deg/sec]", text variable: m_Instance.pMotor1^.stat.lrVelActual
        Label (28,117 70x15), "Initialised"
        Label (28,97 70x15), "Enabled"
        Ellipse (15,118 10x10), tooltip "GREEN=Initialised RED=NOT Initialised", colour toggle: (m_Instance.pMotor1^.stat.bInitialised) <> 0
        Label (105,112 70x25), "Actual Vel:"
        Label (227,180 105x20), "Status"
        Label (437,222 105x20), "Error"
        Rectangle (90,220 355x20), "%s", tooltip "Error Description", text variable: m_Instance.pMotor1^.stat.sErrorText
        Label (28,137 70x15), "Ready"
        Ellipse (15,138 10x10), tooltip "GREEN=Initialised RED=NOT Initialised", colour toggle: (m_Instance.pMotor1^.stat.bAxisReady) <> 0
        Rectangle (90,200 355x20), "%s", tooltip "Motor Status", text variable: m_Instance.pMotor1^.stat.sStatus
        Rectangle (445,200 90x20), "%d", tooltip "Error ID", text variable: m_Instance.pMotor1^.stat.nErrorCode
        Label (94,132 81x25), "Default Vel:"
        Rectangle (180,134 70x20), "%.3f", tooltip "[deg/sec]", text variable: m_Instance.pMotor1^.cfg.lrDefaultVelocity
        Rectangle (80,35 165x25), "%s", text variable: m_Instance.pMotor1^.stat.sState
        Label (12,55 67x30), "Substate:"
        Rectangle (90,245 355x20), "%s", tooltip "Motor Status", text variable: m_Instance.pMotor2^.stat.sStatus
        Label (29,35 46x30), "State:"
        Label (437,267 105x20), "Error"
        Rectangle (354,35 165x25), "%s", text variable: m_Instance.pMotor2^.stat.sState
        Rectangle (80,60 165x25), "%s", text variable: m_Instance.pMotor1^.stat.sSubstate
        Rectangle (354,60 165x25), "%s", text variable: m_Instance.pMotor2^.stat.sSubstate
        Label (287,57 67x30), "Substate:"
        Label (308,34 45x30), "State:"
        Label (136,13 55x25), "Axis1"
        Label (408,13 53x25), "Axis2"
        Label (26,207 55x25), "Axis1"
        Ellipse (15,99 10x10), tooltip "GREEN=Enabled RED=NOT Enabled", colour toggle: (m_Instance.pMotor1^.stat.bEnabled) <> 0
        Ellipse (291,118 10x10), tooltip "GREEN=Initialised RED=NOT Initialised", colour toggle: (m_Instance.pMotor2^.stat.bInitialised) <> 0
        Label (105,152 70x25), "Max Vel:"
        Label (381,152 70x25), "Max Vel:"
    GroupBox (8,14 549x220), "ADC Status"
        Label (10,26 69x27), "Mode:"
        Ellipse (77,83 12x11), tooltip "Engineering Mode: WHITE=Not active GREEN=Activated", colour toggle: (m_Instance.stat.nMode) = E_ADC_MODE.ENG
        Ellipse (77,31 12x12), tooltip "Stationary Mode: WHITE=Not Active GREEN=Activated", colour toggle: (m_Instance.stat.nMode) = E_ADC_MODE.OFF
        Label (92,80 35x18), "ENG"
        Ellipse (77,53 12x12), tooltip "Sky Mode: WHITE=Not Active GREEN=Activated", colour toggle: (m_Instance.stat.nMode) = E_ADC_MODE.AUTO
        Label (92,28 90x20), "OFF"
        Label (310,143 40x20), "Ra:"
        Label (313,162 40x20), "Dec:"
        Rectangle (355,143 95x20), "%.1f", tooltip "TEL RA", text variable: m_Instance.stat.apparent.alpha
        Rectangle (355,163 95x20), "%.1f", tooltip "TEL Dec", text variable: m_Instance.stat.apparent.delta
        Rectangle (490,194 50x20), "%.2f", tooltip "Parallactic Angle [deg]", text variable: m_Instance.stat.data.pa_deg
        Label (437,193 50x20), "PA :"
        Rectangle (491,144 50x20), "%.2f", tooltip "TEL Altitude [deg]", text variable: m_Instance.stat.data.alt_deg
        Rectangle (491,164 50x20), "%.2f", tooltip "TEL Azimuth [deg]", text variable: m_Instance.stat.data.az_deg
        Label (438,143 50x20), "Alt :"
        Label (438,163 50x20), "Az :"
        Rectangle (324,76 218x25), "%s", text variable: m_Instance.stat.sm.sSubstate
        Rectangle (166,76 153x25), "%s", text variable: m_Instance.stat.sm.sState
        Rectangle (166,101 376x25), "%s", text variable: m_Instance.stat.sStatus
        Label (193,50 45x30), "State:"
        Rectangle (392,21 150x20), "Motor.library ver. %s", text variable: m_Instance.stat.sLibVersion
        Rectangle (229,16 150x30), "%s", text variable: m_DeviceName
        Label (389,50 64x30), "Substate:"
        Rectangle (56,143 100x36), "%.1f", text variable: m_Instance.pMotor1^.stat.lrPosActual
        Label (6,179 47x28), "Target"
        Rectangle (56,183 101x20), "%.1f", tooltip "Motor 1 target position in user units (UU).", text variable: m_Instance.pMotor1^.stat.lrPosTarget
        Label (7,148 47x28), "Actual"
        Label (92,50 45x20), "AUTO"
        Rectangle (163,143 100x36), "%.1f", text variable: m_Instance.pMotor2^.stat.lrPosActual
        Rectangle (163,183 101x20), "%.1f", tooltip "Motor 2 target position in user units (UU).", text variable: m_Instance.pMotor2^.stat.lrPosTarget
    Label (447,721 105x20), "Error"
    Rectangle (99,741 355x20), "%s", tooltip "Error Description", text variable: m_Instance.pMotor2^.stat.sErrorText
    Label (37,729 55x25), "Axis2"
    Rectangle (454,721 90x20), "%d", tooltip "Error ID", text variable: m_Instance.pMotor2^.stat.nErrorCode
    Label (382,569 78x25), "Actual Pos:"
    Rectangle (465,570 70x20), "%.3f", tooltip "[deg]", text variable: m_Instance.pMotor2^.stat.lrPosActual
    Rectangle (465,590 70x20), "%.3f", tooltip "[deg/sec]", text variable: m_Instance.pMotor2^.stat.lrVelActual
    Label (313,593 70x15), "Initialised"
    Label (313,573 70x15), "Enabled"
    Label (390,588 70x25), "Actual Vel:"
    Label (313,613 70x15), "Ready"
    Label (377,607 83x25), "Default Vel:"
    Rectangle (465,610 70x20), "%.3f", tooltip "[deg/sec]", text variable: m_Instance.pMotor2^.cfg.lrDefaultVelocity
    Ellipse (300,614 10x10), tooltip "GREEN=Initialised RED=NOT Initialised", colour toggle: (m_Instance.pMotor2^.stat.bAxisReady) <> 0
    Ellipse (300,575 10x10), tooltip "GREEN=Enabled RED=NOT Enabled", colour toggle: (m_Instance.pMotor2^.stat.bEnabled) <> 0
    Rectangle (44,361 70x25), "%.2f", tooltip "ADC2 ENG position angle [deg]", text variable: m_Instance.ctrl.lrTargetPos[2]
        OnMouseDown: write the text variable via Edit
    Rectangle (189,630 70x20), "%.3f", tooltip "[deg/sec]", text variable: m_Instance.pMotor1^.stat.axis.lrMaxVelocity
    Rectangle (465,630 70x20), "%.3f", tooltip "[deg/sec]", text variable: m_Instance.pMotor2^.stat.axis.lrMaxVelocity
END_VISUALIZATION

// VISUs/Templates/GUI_TEMPLATE_MA_DROT
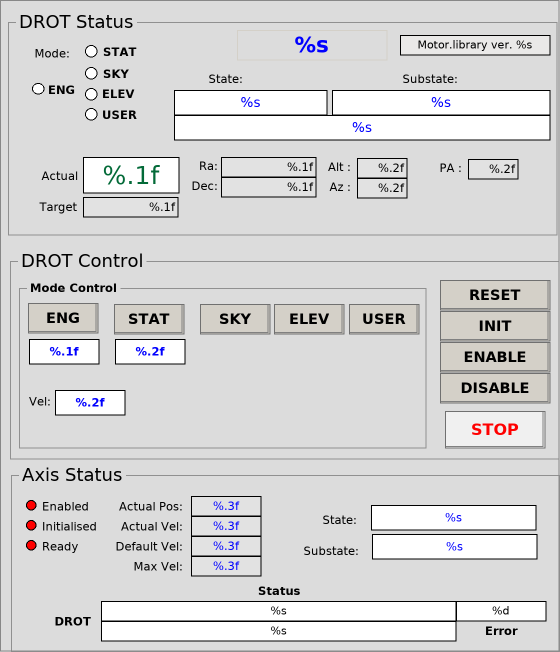
VISUALIZATION GUI_TEMPLATE_MA_DROT  // 560x652
VAR_INPUT
	m_DeviceName : STRING;
END_VAR
VAR_IN_OUT
	m_Instance : FB_MA_DROT;
END_VAR
    GroupBox (10,253 549x206), "DROT Control"
        Button (435,158 100x37), "STOP"
            OnMouseClick: execute { m_Instance.ctrl.nCommand:= E_MA_COMMAND.STOP; m_Instance.ctrl.bExecute:=(TRUE); }
        GroupBox (9,27 407x168), "Mode Control"
            Button (181,24 70x30), "SKY", tooltip "SKY mode (2)"
                OnMouseClick: execute {
                    m_Instance.ctrl.nMode:= E_DROT_MODE.SKY;
                    m_Instance.ctrl.nCommand:=E_MA_COMMAND.START_TRACK;
                    m_Instance.ctrl.bExecute:=(TRUE);
                }
            Rectangle (10,59 70x25), "%.1f", tooltip "[deg]", text variable: m_Instance.ctrl.lrTargetPos
                OnMouseDown: write the text variable via Edit
            Button (9,23 70x30), "ENG", tooltip "Engineering mode (0)"
                OnMouseClick: execute {
                    m_Instance.ctrl.nMode:= E_DROT_MODE.ENG;
                    m_Instance.ctrl.nCommand:= E_MA_COMMAND.STOP_TRACK;
                    m_Instance.ctrl.bExecute:=(TRUE);
                }
            Rectangle (36,110 70x25), "%.2f", tooltip "Velocity for Engineering Mode [deg/sec]", text variable: m_Instance.ctrl.lrTargetVel
                OnMouseDown: write the text variable via Edit
            Button (255,24 70x30), "ELEV", tooltip "ELEV mode (3)"
                OnMouseClick: execute {
                    m_Instance.ctrl.nMode:= E_DROT_MODE.ELEV;
                    m_Instance.ctrl.nCommand:=E_MA_COMMAND.START_TRACK;
                    m_Instance.ctrl.bExecute:=(TRUE);
                }
            Button (95,24 70x30), "STAT", tooltip "STAT mode (1)"
                OnMouseClick: execute {
                    m_Instance.ctrl.nMode:=E_DROT_MODE.STAT;
                    m_Instance.ctrl.nCommand:= E_MA_COMMAND.STOP_TRACK;
                    m_Instance.ctrl.bExecute:=(TRUE);
                }
            Button (330,24 70x30), "USER", tooltip "USER mode (4)"
                OnMouseClick: execute {
                    m_Instance.ctrl.nMode:= E_DROT_MODE.USER;
                    m_Instance.ctrl.nCommand:=E_MA_COMMAND.START_TRACK;
                    m_Instance.ctrl.bExecute:=(TRUE);
                }
            Label (5,109 30x25), "Vel:"
            Rectangle (96,59 70x25), "%.2f", tooltip "Position angle [deg]", text variable: m_Instance.ctrl.lrPosang
                OnMouseDown: write the text variable via Edit
        Button (430,120 110x30), "DISABLE"
            OnMouseClick: execute { m_Instance.ctrl.nCommand:= E_MA_COMMAND.DISABLE; m_Instance.ctrl.bExecute:=(TRUE); }
        Button (430,27 110x30), "RESET"
            OnMouseClick: execute { m_Instance.ctrl.nCommand:= E_MA_COMMAND.RESET; m_Instance.ctrl.bExecute:=(TRUE); }
        Button (430,89 110x30), "ENABLE"
            OnMouseClick: execute { m_Instance.ctrl.nCommand:= E_MA_COMMAND.ENABLE; m_Instance.ctrl.bExecute:=(TRUE); }
        Button (430,58 110x30), "INIT"
            OnMouseClick: execute { m_Instance.ctrl.nCommand:= E_MA_COMMAND.INIT; m_Instance.ctrl.bExecute:=(TRUE); }
    GroupBox (11,467 549x185), "Axis Status"
        Label (105,27 70x25), "Actual Pos:"
        Rectangle (180,29 70x20), "%.3f", tooltip "[deg]", text variable: m_Instance.pMotor1^.stat.lrPosActual
        Rectangle (180,49 70x20), "%.3f", tooltip "[deg/sec]", text variable: m_Instance.pMotor1^.stat.lrVelActual
        Label (28,52 70x15), "Initialised"
        Ellipse (15,33 10x10), tooltip "GREEN=Enabled RED=NOT Enabled", colour toggle: (m_Instance.pMotor1^.stat.bEnabled) <> 0
        Label (28,32 70x15), "Enabled"
        Ellipse (15,53 10x10), tooltip "GREEN=Initialised RED=NOT Initialised", colour toggle: (m_Instance.pMotor1^.stat.bInitialised) <> 0
        Label (105,47 70x25), "Actual Vel:"
        Label (216,114 105x20), "Status"
        Label (438,154 105x20), "Error"
        Rectangle (90,154 355x20), "%s", tooltip "Error Description", text variable: m_Instance.pMotor1^.stat.sErrorText
        Label (28,142 55x25), "DROT"
        Label (28,72 70x15), "Ready"
        Ellipse (15,73 10x10), tooltip "GREEN=Initialised RED=NOT Initialised", colour toggle: (m_Instance.pMotor1^.stat.bAxisReady) <> 0
        Rectangle (90,134 355x20), "%s", tooltip "Motor Status", text variable: m_Instance.pMotor1^.stat.sStatus
        Rectangle (445,134 90x20), "%d", tooltip "Error ID", text variable: m_Instance.pMotor1^.stat.nErrorCode
        Label (105,67 70x25), "Default Vel:"
        Rectangle (180,69 70x20), "%.3f", tooltip "[deg/sec]", text variable: m_Instance.pMotor1^.cfg.lrDefaultVelocity
        Rectangle (360,38 165x25), "%s", text variable: m_Instance.pMotor1^.stat.sState
        Label (259,38 90x30), "State:"
        Label (261,69 90x30), "Substate:"
        Rectangle (361,67 165x25), "%s", text variable: m_Instance.pMotor1^.stat.sSubstate
        Label (105,87 70x25), "Max Vel:"
        Rectangle (180,89 70x20), "%.3f", tooltip "[deg/sec]", text variable: m_Instance.pMotor1^.stat.axis.lrMaxVelocity
    GroupBox (8,14 549x221), "DROT Status"
        Label (10,26 69x27), "Mode:"
        Ellipse (24,69 12x11), tooltip "Engineering Mode: WHITE=Not active GREEN=Activated", colour toggle: (m_Instance.stat.nMode) = E_DROT_MODE.ENG
        Ellipse (77,31 12x12), tooltip "Stationary Mode: WHITE=Not Active GREEN=Activated", colour toggle: (m_Instance.stat.nMode) = E_DROT_MODE.STAT
        Label (37,67 83x18), "ENG"
        Ellipse (77,53 12x12), tooltip "Sky Mode: WHITE=Not Active GREEN=Activated", colour toggle: (m_Instance.stat.nMode) = E_DROT_MODE.SKY
        Ellipse (77,74 12x12), tooltip "Elevation Mode: WHITE=Not Active GREEN=Activated", colour toggle: (m_Instance.stat.nMode) = E_DROT_MODE.ELEV
        Label (91,70 43x20), "ELEV"
        Label (92,50 45x20), "SKY"
        Label (92,28 90x20), "STAT"
        Label (173,142 40x20), "Ra:"
        Label (173,162 40x20), "Dec:"
        Rectangle (213,143 95x20), "%.1f", tooltip "TEL RA", text variable: m_Instance.stat.apparent.alpha
        Rectangle (213,163 95x20), "%.1f", tooltip "TEL Dec", text variable: m_Instance.stat.apparent.delta
        Rectangle (460,145 50x20), "%.2f", tooltip "Parallactic Angle [deg]", text variable: m_Instance.stat.data.pa_deg
        Label (407,144 50x20), "PA :"
        Rectangle (349,144 50x20), "%.2f", tooltip "TEL Altitude [deg]", text variable: m_Instance.stat.data.alt_deg
        Rectangle (349,164 50x20), "%.2f", tooltip "TEL Azimuth [deg]", text variable: m_Instance.stat.data.az_deg
        Label (296,143 50x20), "Alt :"
        Label (296,163 50x20), "Az :"
        Rectangle (324,76 218x25), "%s", text variable: m_Instance.stat.sm.sSubstate
        Rectangle (166,76 153x25), "%s", text variable: m_Instance.stat.sm.sState
        Rectangle (166,101 376x25), "%s", text variable: m_Instance.stat.sStatus
        Label (193,50 45x30), "State:"
        Rectangle (392,21 150x20), "Motor.library ver. %s", text variable: m_Instance.stat.sLibVersion
        Rectangle (229,16 150x30), "%s", text variable: m_DeviceName
        Label (389,50 64x30), "Substate:"
        Rectangle (75,143 96x36), "%.1f", text variable: m_Instance.pMotor1^.stat.lrPosActual
        Label (25,179 47x28), "Target"
        Rectangle (75,183 95x20), "%.1f", tooltip "TEL RA", text variable: m_Instance.stat.lrPos
        Label (26,148 47x28), "Actual"
        Ellipse (77,94 12x12), tooltip "User defined Mode: WHITE=Not Active GREEN=Activated", colour toggle: (m_Instance.stat.nMode) = E_DROT_MODE.USER
        Label (91,91 45x20), "USER"
END_VISUALIZATION

// VISUs/Templates/GUI_TEMPLATE_MOTOR_CONFIG
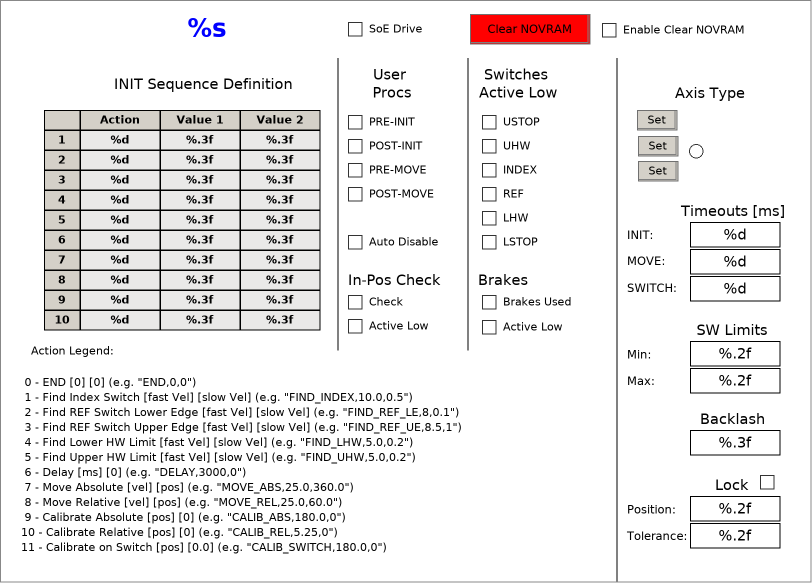
VISUALIZATION GUI_TEMPLATE_MOTOR_CONFIG  // 812x583
VAR_IN_OUT
	m_Instance : FB_MOTOR;
END_VAR
VAR
	bEnableNovramClear:	BOOL := FALSE;
END_VAR
    Label (28,336 150x30), "Action Legend:"
    Label (18,371 600x23), "0 - END [0] [0] (e.g. "END,0,0")"
    Label (18,386 600x23), "1 - Find Index Switch [fast Vel] [slow Vel] (e.g. "FIND_INDEX,10.0,0.5")"
    Label (18,401 600x23), "2 - Find REF Switch Lower Edge [fast Vel] [slow Vel] (e.g. "FIND_REF_LE,8,0.1")"
    Label (18,416 600x23), "3 - Find REF Switch Upper Edge [fast Vel] [slow Vel] (e.g. "FIND_REF_UE,8.5,1")"
    Label (18,431 600x23), "4 - Find Lower HW Limit [fast Vel] [slow Vel] (e.g. "FIND_LHW,5.0,0.2")"
    Label (18,446 600x23), "5 - Find Upper HW Limit [fast Vel] [slow Vel] (e.g. "FIND_UHW,5.0,0.2")"
    Label (18,476 600x23), "7 - Move Absolute [vel] [pos] (e.g. "MOVE_ABS,25.0,360.0")"
    Label (18,491 600x23), "8 - Move Relative [vel] [pos] (e.g. "MOVE_REL,25.0,60.0")"
    Label (18,506 600x23), "9 - Calibrate Absolute [pos] [0] (e.g. "CALIB_ABS,180.0,0")"
    Label (18,521 600x23), "10 - Calibrate Relative [pos] [0] (e.g. "CALIB_REL,5.25,0")"
    Label (18,461 600x23), "6 - Delay [ms] [0] (e.g. "DELAY,3000,0")"
    Label (18,536 600x23), "11 - Calibrate on Switch [pos] [0.0] (e.g. "CALIB_SWITCH,180.0,0")"
    Label (59,69 289x30), "INIT Sequence Definition"
    Label (462,54 113x59), "Switches Active Low"
    Checkbox (480,110 93x24), "USTOP", variable: m_Instance.cfg.bArrActiveLow[5].bValue, invisible if: false, input disabled if: false
    Checkbox (480,134 93x24), "UHW", variable: m_Instance.cfg.bArrActiveLow[4].bValue, invisible if: false, input disabled if: false
    Checkbox (480,158 93x24), "INDEX", variable: m_Instance.cfg.bArrActiveLow[3].bValue, invisible if: false, input disabled if: false
    Checkbox (480,182 93x24), "REF", variable: m_Instance.cfg.bArrActiveLow[2].bValue, invisible if: false, input disabled if: false
    Checkbox (480,206 93x24), "LHW", variable: m_Instance.cfg.bArrActiveLow[1].bValue, invisible if: false, input disabled if: false
    Checkbox (480,230 93x24), "LSTOP", variable: m_Instance.cfg.bArrActiveLow[0].bValue, invisible if: false, input disabled if: false
    Rectangle (87,7 240x42), "%s", text variable: m_Instance.sName
    Label (678,196 132x30), "Timeouts [ms]"
    Label (665,78 90x30), "Axis Type"
    Label (687,315 90x30), "SW Limits"
    Label (475,265 103x30), "Brakes"
    Label (685,404 95x30), "Backlash"
    RadioButton (687,112 114x78), variable: m_Instance.cfg.nAxisType-1, input disabled if: FALSE
        Areas[0]: Text=Linear
        Areas[1]: Text=Circular
        Areas[2]: Text=Circular-Opt
        p3166011961: Cicular-Optimised
    Checkbox (480,290 110x24), "Brakes Used", variable: m_Instance.cfg.bUseBrake, invisible if: false, input disabled if: false
    Checkbox (480,315 105x24), "Active Low", tooltip "Brake Feedback Signal is Active Low", variable: m_Instance.cfg.bActiveLowBrake, invisible if: false, input disabled if: false
    Rectangle (690,430 90x25), "%.3f", tooltip "Positive, negative or zero (no backlash)", text variable: m_Instance.cfg.lrBacklash
        OnMouseDown: write the text variable via Default
    Button (637,110 40x20), "Set"
        OnMouseClick: execute { m_Instance.cfg.nAxisType := 1; }
    Button (638,136 40x20), "Set"
        OnMouseClick: execute { m_Instance.cfg.nAxisType := 2; }
    Button (638,161 40x20), "Set"
        OnMouseClick: execute { m_Instance.cfg.nAxisType := 3; }
    Rectangle (690,341 90x25), "%.2f", tooltip "Setting both limits to 0 means that limits are not used.", text variable: m_Instance.cfg.lrMinPosition
        OnMouseDown: write the text variable via Default
    Rectangle (690,368 90x25), "%.2f", tooltip "Setting both limits to 0 means that limits are not used.", text variable: m_Instance.cfg.lrMaxPosition
        OnMouseDown: write the text variable via Default
    Label (624,340 37x29), "Min:"
    Label (624,366 37x30), "Max:"
    Label (624,220 49x30), "INIT:"
    Label (624,246 49x30), "MOVE:"
    Rectangle (690,222 90x25), "%d", tooltip "INIT sequence timeout in [ms].", text variable: m_Instance.cfg.nTimeoutInit
        OnMouseDown: write the text variable via Default
    Rectangle (690,249 90x25), "%d", tooltip "INIT sequence timeout in [ms].", text variable: m_Instance.cfg.nTimeoutMove
        OnMouseDown: write the text variable via Default
    Line (468,350) (468,58)
    Line (617,581) (617,58)
    Rectangle (690,276 90x25), "%d", tooltip "Switch exit timeout in [ms].", text variable: m_Instance.cfg.nTimeoutSwitch
        OnMouseDown: write the text variable via Default
    Label (624,273 60x30), "SWITCH:"
    Rectangle (80,110 80x20), "Action"
    Rectangle (160,110 80x20), "Value 1"
    Rectangle (240,110 80x20), "Value 2"
    Rectangle (44,130 36x20), "1"
    Rectangle (44,110 36x20)
    Rectangle (80,130 80x20), "%d", text variable: m_Instance.cfg.strArrInitSeq[1].nAction
        OnMouseDown: write the text variable via Default
    Rectangle (160,130 80x20), "%.3f", text variable: m_Instance.cfg.strArrInitSeq[1].lrValue1
        OnMouseDown: write the text variable via Default
    Rectangle (240,130 80x20), "%.3f", text variable: m_Instance.cfg.strArrInitSeq[1].lrValue2
        OnMouseDown: write the text variable via Default
    Rectangle (44,150 36x20), "2"
    Rectangle (80,150 80x20), "%d", text variable: m_Instance.cfg.strArrInitSeq[2].nAction
        OnMouseDown: write the text variable via Default
    Rectangle (160,150 80x20), "%.3f", text variable: m_Instance.cfg.strArrInitSeq[2].lrValue1
        OnMouseDown: write the text variable via Default
    Rectangle (240,150 80x20), "%.3f", text variable: m_Instance.cfg.strArrInitSeq[2].lrValue2
        OnMouseDown: write the text variable via Default
    Rectangle (44,170 36x20), "3"
    Rectangle (80,170 80x20), "%d", text variable: m_Instance.cfg.strArrInitSeq[3].nAction
        OnMouseDown: write the text variable via Default
    Rectangle (160,170 80x20), "%.3f", text variable: m_Instance.cfg.strArrInitSeq[3].lrValue1
        OnMouseDown: write the text variable via Default
    Rectangle (240,170 80x20), "%.3f", text variable: m_Instance.cfg.strArrInitSeq[3].lrValue2
        OnMouseDown: write the text variable via Default
    Rectangle (44,190 36x20), "4"
    Rectangle (80,190 80x20), "%d", text variable: m_Instance.cfg.strArrInitSeq[4].nAction
        OnMouseDown: write the text variable via Default
    Rectangle (160,190 80x20), "%.3f", text variable: m_Instance.cfg.strArrInitSeq[4].lrValue1
        OnMouseDown: write the text variable via Default
    Rectangle (240,190 80x20), "%.3f", text variable: m_Instance.cfg.strArrInitSeq[4].lrValue2
        OnMouseDown: write the text variable via Default
    Rectangle (44,210 36x20), "5"
    Rectangle (80,210 80x20), "%d", text variable: m_Instance.cfg.strArrInitSeq[5].nAction
        OnMouseDown: write the text variable via Default
    Rectangle (160,210 80x20), "%.3f", text variable: m_Instance.cfg.strArrInitSeq[5].lrValue1
        OnMouseDown: write the text variable via Default
    Rectangle (240,210 80x20), "%.3f", text variable: m_Instance.cfg.strArrInitSeq[5].lrValue2
        OnMouseDown: write the text variable via Default
    Rectangle (44,230 36x20), "6"
    Rectangle (80,230 80x20), "%d", text variable: m_Instance.cfg.strArrInitSeq[6].nAction
        OnMouseDown: write the text variable via Default
    Rectangle (160,230 80x20), "%.3f", text variable: m_Instance.cfg.strArrInitSeq[6].lrValue1
        OnMouseDown: write the text variable via Default
    Rectangle (240,230 80x20), "%.3f", text variable: m_Instance.cfg.strArrInitSeq[6].lrValue2
        OnMouseDown: write the text variable via Default
    Rectangle (44,250 36x20), "7"
    Rectangle (80,250 80x20), "%d", text variable: m_Instance.cfg.strArrInitSeq[7].nAction
        OnMouseDown: write the text variable via Default
    Rectangle (160,250 80x20), "%.3f", text variable: m_Instance.cfg.strArrInitSeq[7].lrValue1
        OnMouseDown: write the text variable via Default
    Rectangle (240,250 80x20), "%.3f", text variable: m_Instance.cfg.strArrInitSeq[7].lrValue2
        OnMouseDown: write the text variable via Default
    Rectangle (44,270 36x20), "8"
    Rectangle (80,270 80x20), "%d", text variable: m_Instance.cfg.strArrInitSeq[8].nAction
        OnMouseDown: write the text variable via Default
    Rectangle (160,270 80x20), "%.3f", text variable: m_Instance.cfg.strArrInitSeq[8].lrValue1
        OnMouseDown: write the text variable via Default
    Rectangle (240,270 80x20), "%.3f", text variable: m_Instance.cfg.strArrInitSeq[8].lrValue2
        OnMouseDown: write the text variable via Default
    Rectangle (44,290 36x20), "9"
    Rectangle (80,290 80x20), "%d", text variable: m_Instance.cfg.strArrInitSeq[9].nAction
        OnMouseDown: write the text variable via Default
    Rectangle (160,290 80x20), "%.3f", text variable: m_Instance.cfg.strArrInitSeq[9].lrValue1
        OnMouseDown: write the text variable via Default
    Rectangle (240,290 80x20), "%.3f", text variable: m_Instance.cfg.strArrInitSeq[9].lrValue2
        OnMouseDown: write the text variable via Default
    Rectangle (44,310 36x20), "10"
    Rectangle (80,310 80x20), "%d", text variable: m_Instance.cfg.strArrInitSeq[10].nAction
        OnMouseDown: write the text variable via Default
    Rectangle (160,310 80x20), "%.3f", text variable: m_Instance.cfg.strArrInitSeq[10].lrValue1
        OnMouseDown: write the text variable via Default
    Rectangle (240,310 80x20), "%.3f", text variable: m_Instance.cfg.strArrInitSeq[10].lrValue2
        OnMouseDown: write the text variable via Default
    Line (338,350) (338,58)
    Label (345,54 94x59), "User Procs"
    Checkbox (346,110 106x24), "PRE-INIT", variable: m_Instance.cfg.bExecUserPreInit, invisible if: false, input disabled if: false
    Checkbox (346,134 106x24), "POST-INIT", variable: m_Instance.cfg.bExecUserPostInit, invisible if: false, input disabled if: false
    Checkbox (346,158 106x24), "PRE-MOVE", variable: m_Instance.cfg.bExecUserPreMove, invisible if: false, input disabled if: false
    Checkbox (346,182 106x24), "POST-MOVE", variable: m_Instance.cfg.bExecUserPostMove, invisible if: false, input disabled if: false
    Label (687,470 90x30), "Lock"
    Rectangle (690,496 90x25), "%.2f", tooltip "If the motor is locked, during INIT the motor will not move and its position will be set to this value.", text variable: m_Instance.cfg.lrLockPos
        OnMouseDown: write the text variable via Default
    Rectangle (690,523 90x25), "%.2f", tooltip "The motor will not move, if the target position is closer to the locked position than this value.", text variable: m_Instance.cfg.lrLockTol
        OnMouseDown: write the text variable via Default
    Label (624,495 56x29), "Position:"
    Label (624,521 63x30), "Tolerance:"
    Checkbox (758,470 30x24), tooltip "Flag if motor is locked", variable: m_Instance.cfg.bLock, invisible if: false, input disabled if: false
    Checkbox (346,290 106x24), "Check", tooltip "If active, check if the in-pos signal is active after the move completes. If it is not, it's a failure.", variable: m_Instance.cfg.bCheckInPos, invisible if: false, input disabled if: false
    Checkbox (346,314 107x24), "Active Low", tooltip "If checked, In-Position feedback signal is active low", variable: m_Instance.cfg.bActiveLowInPos, invisible if: false, input disabled if: false
    Checkbox (346,230 127x24), "Auto Disable", tooltip "Auto Disable Motor After Move", variable: m_Instance.cfg.bDisableAfterMove, invisible if: false, input disabled if: false
    Label (345,265 103x30), "In-Pos Check"
    Button (470,14 120x30), "Clear NOVRAM", tooltip "Clear NOVRAM. Use it with care! This is needed ONLY if NOVRAM was previously used for data structures different than T_MOTOR_CFG (or for previous versions of T_MOTOR_CFG). Bring the motor to NOT_READY first and then clear NOVRAM.", input disabled if: bEnableNovramClear=false OR m_Instance.nNOVRAM_DevId=0
        OnMouseUp: execute {
            m_Instance.ctrl.bLocalCmd := TRUE;
            m_Instance.ctrl.nCommand:=E_MOTOR_COMMAND.CLEAR_NOVRAM;
            m_Instance.ctrl.bExecute:=(TRUE);
        }
    Checkbox (600,18 160x24), "Enable Clear NOVRAM", variable: bEnableNovramClear, invisible if: false, input disabled if: false
    Checkbox (346,17 90x24), "SoE Drive", tooltip "Check the box if this is an SoE drive (Sercos over EtherCAT) , e.g. AX5000", variable: m_Instance.cfg.bSoE_Drive, invisible if: false, input disabled if: false
END_VISUALIZATION

// VISUs/Templates/GUI_TEMPLATE_MOTOR_CONTROL
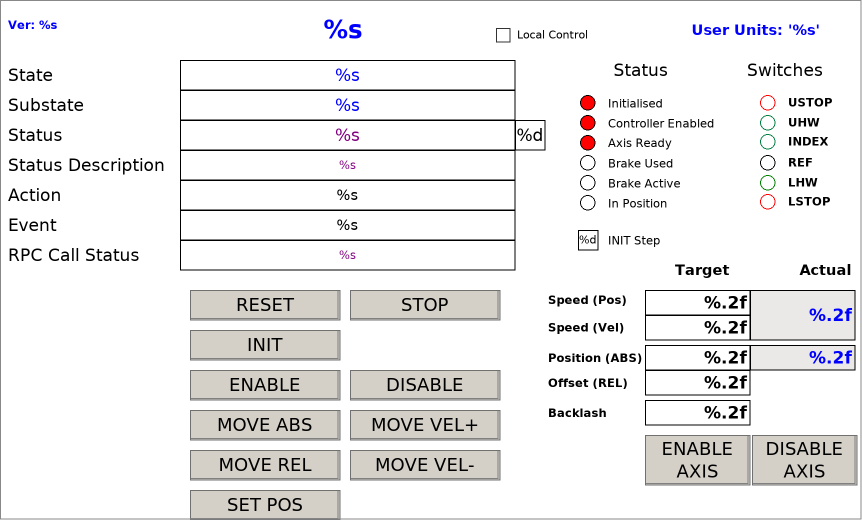
VISUALIZATION GUI_TEMPLATE_MOTOR_CONTROL  // 862x520
VAR_IN_OUT
	m_Instance:	FB_MOTOR;
END_VAR
    Rectangle (180,60 335x30), "%s", text variable: m_Instance.stat.sState
    Rectangle (180,90 335x30), "%s", text variable: m_Instance.stat.sSubstate
    Button (190,290 150x30), "RESET", input disabled if: (m_Instance.stat.bLocal = FALSE) <> 0
        OnMouseDown: execute {
            m_Instance.ctrl.bLocalCmd := TRUE;
            m_Instance.ctrl.nCommand := E_MOTOR_COMMAND.RESET;
            m_Instance.ctrl.bExecute := TRUE;
        }
    Button (190,330 150x30), "INIT", input disabled if: (m_Instance.stat.bLocal = FALSE) <> 0
        OnMouseDown: execute {
            m_Instance.ctrl.bLocalCmd := TRUE;
            m_Instance.ctrl.nCommand := E_MOTOR_COMMAND.INIT;
            m_Instance.ctrl.bExecute := TRUE;
        }
    Button (350,290 150x30), "STOP", input disabled if: (m_Instance.stat.bLocal = FALSE) <> 0
        OnMouseDown: execute {
            m_Instance.ctrl.bLocalCmd := TRUE;
            m_Instance.ctrl.nCommand := E_MOTOR_COMMAND.STOP;
            m_Instance.ctrl.bExecute := TRUE;
        }
    Button (190,370 150x30), "ENABLE", input disabled if: (m_Instance.stat.bLocal = FALSE) <> 0
        OnMouseDown: execute {
            m_Instance.ctrl.bLocalCmd := TRUE;
            m_Instance.ctrl.nCommand := E_MOTOR_COMMAND.ENABLE;
            m_Instance.ctrl.bExecute := TRUE;
        }
    Button (350,370 150x30), "DISABLE", input disabled if: (m_Instance.stat.bLocal = FALSE) <> 0
        OnMouseDown: execute {
            m_Instance.ctrl.bLocalCmd := TRUE;
            m_Instance.ctrl.nCommand := E_MOTOR_COMMAND.DISABLE;
            m_Instance.ctrl.bExecute := TRUE;
        }
    Button (190,410 150x30), "MOVE ABS", input disabled if: (m_Instance.stat.bLocal = FALSE) <> 0
        OnMouseDown: execute {
            m_Instance.ctrl.bLocalCmd := TRUE;
            m_Instance.ctrl.lrVelocity:=(m_Instance.cfg.lrDefaultVelocity);
            m_Instance.ctrl.nCommand := E_MOTOR_COMMAND.MOTOR_MOVE;
            m_Instance.ctrl.nMoveType := E_MOTOR_MOVE_TYPE.ABSOLUTE;
            m_Instance.ctrl.bExecute := TRUE;
        }
    Button (350,410 150x30), "MOVE VEL+", input disabled if: (m_Instance.stat.bLocal = FALSE) <> 0
        OnMouseDown: execute {
            m_Instance.ctrl.bLocalCmd := TRUE;
            m_Instance.ctrl.nCommand := E_MOTOR_COMMAND.MOTOR_MOVE;
            m_Instance.ctrl.nMoveType := E_MOTOR_MOVE_TYPE.VELOCITY;
            m_Instance.ctrl.nDirection := MC_Positive_Direction;
            m_Instance.ctrl.bExecute := TRUE;
        }
    Rectangle (5,60 170x30), "State"
    Rectangle (5,90 170x30), "Substate"
    Rectangle (180,120 335x30), "%s", text variable: m_Instance.stat.sStatus
    Rectangle (180,150 335x30), "%s", tooltip "Additional information mostly used for description of errors", text variable: m_Instance.stat.sErrorText
    Rectangle (5,120 170x30), "Status"
    Rectangle (5,150 170x30), "Status Description"
    Rectangle (180,180 335x30), "%s", text variable: m_Instance.stat.sActionDesc
    Rectangle (180,210 335x30), "%s", text variable: m_Instance.stat.sEventDesc
    Rectangle (5,180 170x30), "Action"
    Rectangle (5,210 170x30), "Event"
    Rectangle (227,12 232x35), "%s", text variable: m_Instance.sName
    Checkbox (494,20 116x30), "Local Control", variable: m_Instance.stat.bLocal
    Rectangle (595,55 92x30), "Status"
    Rectangle (515,120 30x30), "%d", text variable: m_Instance.stat.nStatus
    Rectangle (739,55 92x30), "Switches"
    Button (350,450 150x30), "MOVE VEL-", input disabled if: (m_Instance.stat.bLocal = FALSE) <> 0
        OnMouseDown: execute {
            m_Instance.ctrl.bLocalCmd := TRUE;
            m_Instance.ctrl.nCommand := E_MOTOR_COMMAND.MOTOR_MOVE;
            m_Instance.ctrl.nMoveType := E_MOTOR_MOVE_TYPE.VELOCITY;
            m_Instance.ctrl.nDirection := MC_Negative_Direction;
            m_Instance.ctrl.bExecute := TRUE;
        }
    Button (190,450 150x30), "MOVE REL", input disabled if: (m_Instance.stat.bLocal = FALSE) <> 0
        OnMouseDown: execute {
            m_Instance.ctrl.bLocalCmd := TRUE;
            m_Instance.ctrl.lrVelocity:=(m_Instance.cfg.lrDefaultVelocity);
            m_Instance.ctrl.nCommand := E_MOTOR_COMMAND.MOTOR_MOVE;
            m_Instance.ctrl.nMoveType := E_MOTOR_MOVE_TYPE.RELATIVE;
            m_Instance.ctrl.bExecute := TRUE;
        }
    Button (190,490 150x30), "SET POS", input disabled if: (m_Instance.stat.bLocal = FALSE) <> 0
        OnMouseDown: execute {
            m_Instance.ctrl.bLocalCmd := TRUE;
            m_Instance.ctrl.nCommand := E_MOTOR_COMMAND.SET_POSITION;
            m_Instance.ctrl.bExecute := TRUE;
        }
    Rectangle (785,95 50x15), "USTOP"
    Ellipse (760,95 15x15), colour toggle: m_Instance.stat.signals[5].bActive
    Ellipse (760,115 15x15), colour toggle: m_Instance.stat.signals[4].bActive
    Ellipse (760,175 15x15), colour toggle: m_Instance.stat.signals[1].bActive
    Ellipse (760,194 15x15), colour toggle: m_Instance.stat.signals[0].bActive
    Ellipse (760,155 15x15), colour toggle: m_Instance.stat.signals[2].bActive
    Rectangle (785,134 50x15), "INDEX"
    Rectangle (785,115 50x15), "UHW"
    Rectangle (785,155 50x15), "REF"
    Rectangle (785,175 50x15), "LHW"
    Rectangle (785,194 50x15), "LSTOP"
    Ellipse (760,134 15x15), colour toggle: m_Instance.stat.signals[3].bActive
    Rectangle (545,290 95x20), "Speed (Pos)"
    Rectangle (750,345 105x25), "%.2f", text variable: m_Instance.stat.lrPosActual, input disabled if: false
    Rectangle (672,260 190x20), "Target Actual"
    Rectangle (545,348 95x20), "Position (ABS)"
    Rectangle (750,290 105x50), "%.2f", text variable: m_Instance.stat.lrVelActual, input disabled if: false
    Rectangle (645,315 105x25), "%.2f", text variable: m_Instance.ctrl.lrVelocity
        OnMouseDown: write the text variable via Default
    Rectangle (545,403 95x20), "Backlash"
    Rectangle (645,400 105x25), "%.2f", text variable: m_Instance.cfg.lrBacklash
        OnMouseDown: write the text variable via Default
    Rectangle (545,315 95x25), "Speed (Vel)"
    Rectangle (645,345 105x25), "%.2f", tooltip "Absolute position used by "MOVE ABS"", text variable: m_Instance.ctrl.lrPosition
        OnMouseDown: write the text variable via Default
    Rectangle (645,290 105x25), "%.2f", text variable: m_Instance.cfg.lrDefaultVelocity
        OnMouseDown: write the text variable via Default
    Rectangle (605,171 90x25), "Brake Active"
    Ellipse (580,175 15x15), tooltip "RED = Applied BLANK = Released", colour toggle: (m_Instance.stat.bBrakeActive) <> 0
    Ellipse (580,95 15x15), tooltip "GREEN = Initialised RED = Not Initialised", text variable: m_Instance.stat.bInitialised, colour toggle: m_Instance.stat.bInitialised
    Rectangle (605,91 90x25), "Initialised"
    Rectangle (605,111 125x25), "Controller Enabled"
    Rectangle (605,131 90x24), "Axis Ready"
    Rectangle (605,151 90x25), "Brake Used"
    Ellipse (580,115 15x15), tooltip "GREEN = Enabled RED = Disabled", colour toggle: m_Instance.stat.bEnabled
    Ellipse (580,135 15x15), tooltip "GREEN = Ready RED = Not Ready", colour toggle: m_Instance.stat.bAxisReady
    Ellipse (580,155 15x15), tooltip "BLUE = Used BLANK = Not Used", colour toggle: m_Instance.cfg.bUseBrake
    Rectangle (578,230 20x20), "%d", text variable: m_Instance.stat.nInitStep
    Rectangle (605,228 90x25), "INIT Step"
    Rectangle (5,240 170x30), "RPC Call Status"
    Rectangle (180,240 335x30), "%s", text variable: m_Instance.stat.sRPCErrorText
    Rectangle (605,191 90x25), "In Position"
    Ellipse (580,195 15x15), tooltip "GREEN = In Position BLANK = Not In Position (or not used)", colour toggle: (m_Instance.stat.bInPosition) <> 0
    Button (645,435 105x50), "ENABLE AXIS", input disabled if: (m_Instance.stat.bLocal = FALSE) <> 0
        OnMouseDown: execute { m_Instance.stat.bEnabled := TRUE; }
    Button (752,435 105x50), "DISABLE AXIS", input disabled if: (m_Instance.stat.bLocal = FALSE) <> 0
        OnMouseDown: execute { m_Instance.stat.bEnabled := FALSE; }
    Rectangle (620,15 203x30), "User Units: '%s'", text variable: m_Instance.stat.axis.sUnits
    Rectangle (5,10 99x30), "Ver: %s", tooltip "'Motor.library version'", text variable: m_Instance.stat.sLibVersion, input disabled if: true
    Rectangle (545,373 95x20), "Offset (REL)"
    Rectangle (645,370 105x25), "%.2f", tooltip "Relative offset used by "MOVE REL"", text variable: m_Instance.ctrl.lrOffset
        OnMouseDown: write the text variable via Default
END_VISUALIZATION

// VISUs/Tracking/GUI_ADC_Motor1
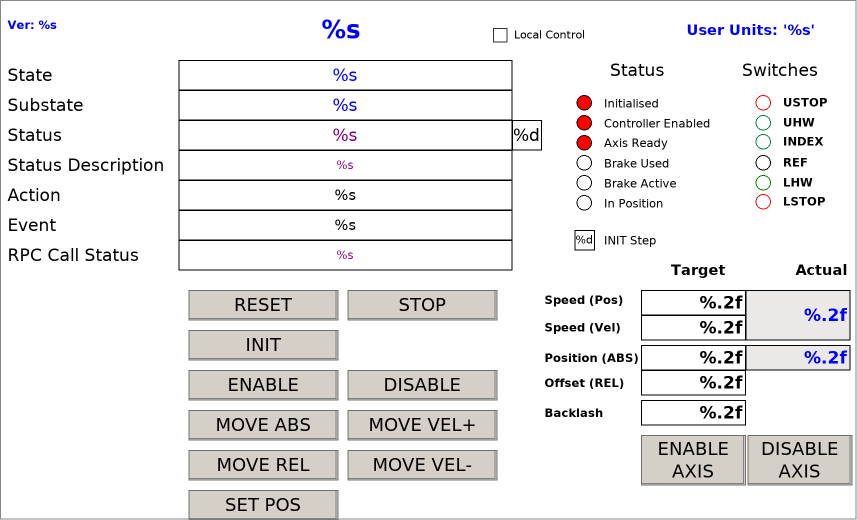
VISUALIZATION GUI_ADC_Motor1  // 857x520
    Frame (0,0 857x520)
        shows GUI_TEMPLATE_MOTOR_CONTROL(m_Instance := MAIN.adc.motor1)
END_VISUALIZATION

// VISUs/Tracking/GUI_ADC_Motor2
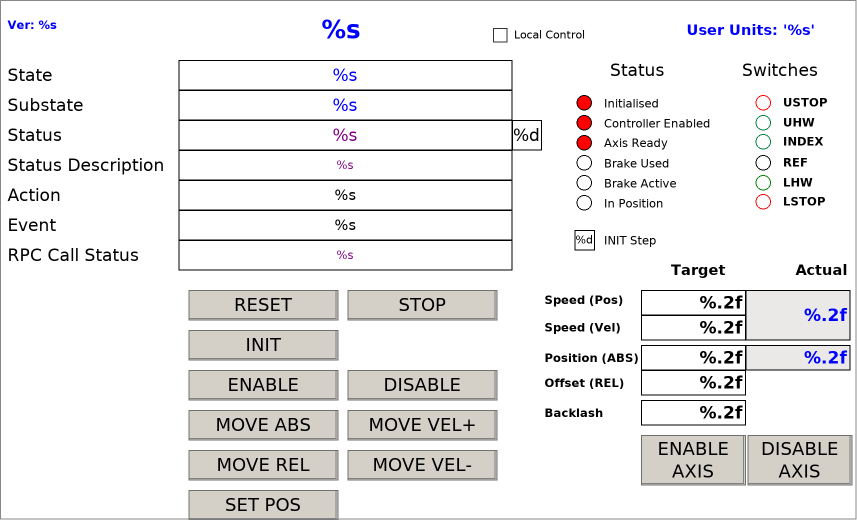
VISUALIZATION GUI_ADC_Motor2  // 857x520
    Frame (0,0 857x520)
        shows GUI_TEMPLATE_MOTOR_CONTROL(m_Instance := MAIN.adc.motor2)
END_VISUALIZATION

// VISUs/Tracking/GUI_CCS_SIM
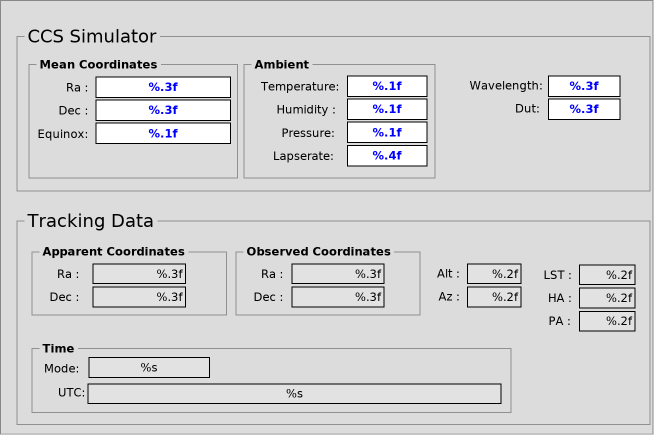
VISUALIZATION GUI_CCS_SIM  // 654x435
    Frame (0,0 652x433)
        shows GUI_TEMPLATE_CCS_SIM(m_DeviceName := 'CCS SIM', m_Instance := MAIN.ccs_sim)
END_VISUALIZATION

// VISUs/Tracking/GUI_DROT_Cfg
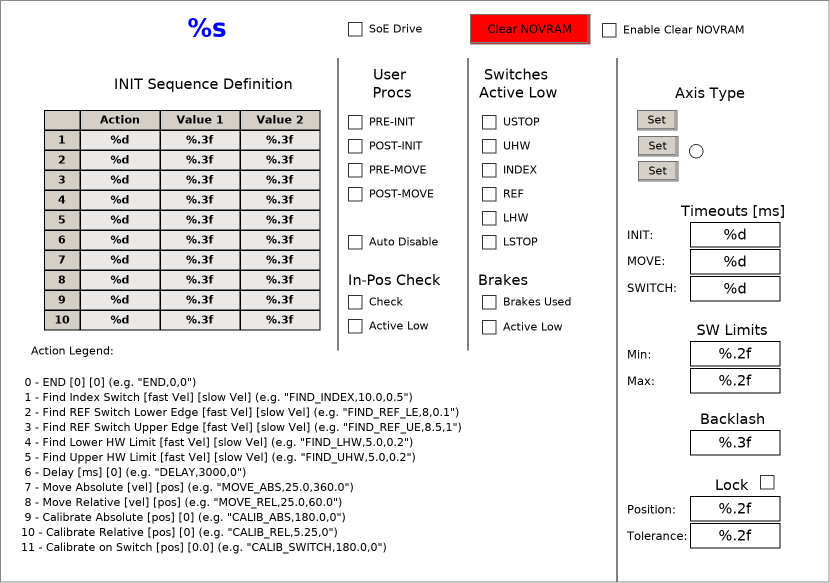
VISUALIZATION GUI_DROT_Cfg  // 830x583
    Frame (0,0 828x581)
        shows GUI_TEMPLATE_MOTOR_CONFIG(m_Instance := MAIN.drot.motor)
END_VISUALIZATION

// VISUs/Tracking/GUI_DROT_Motor
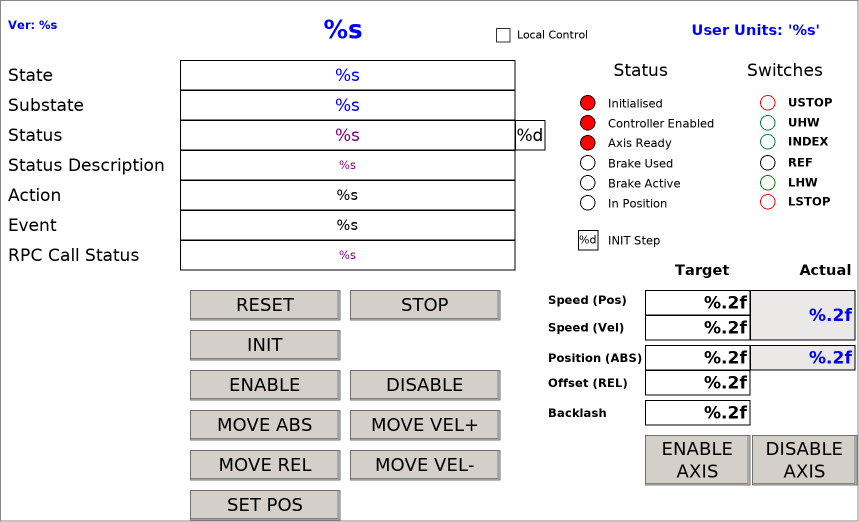
VISUALIZATION GUI_DROT_Motor  // 859x522
    Frame (0,0 857x520)
        shows GUI_TEMPLATE_MOTOR_CONTROL(m_Instance := MAIN.drot.motor)
END_VISUALIZATION

// VISUs/Tracking/GUI_MA_ADC
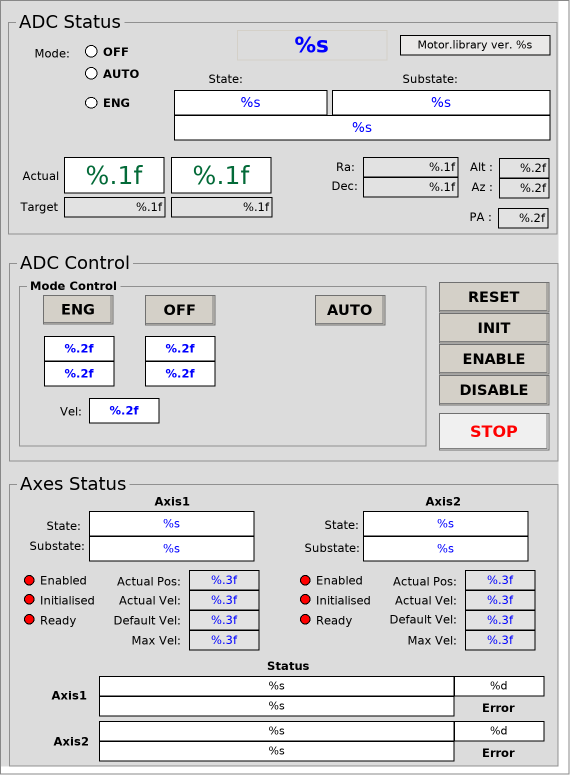
VISUALIZATION GUI_MA_ADC  // 570x775
    Frame (0,0 568x773)
        shows GUI_TEMPLATE_MA_ADC(m_DeviceName := 'ADC', m_Instance := MAIN.adc)
END_VISUALIZATION

// VISUs/Tracking/GUI_MA_DROT
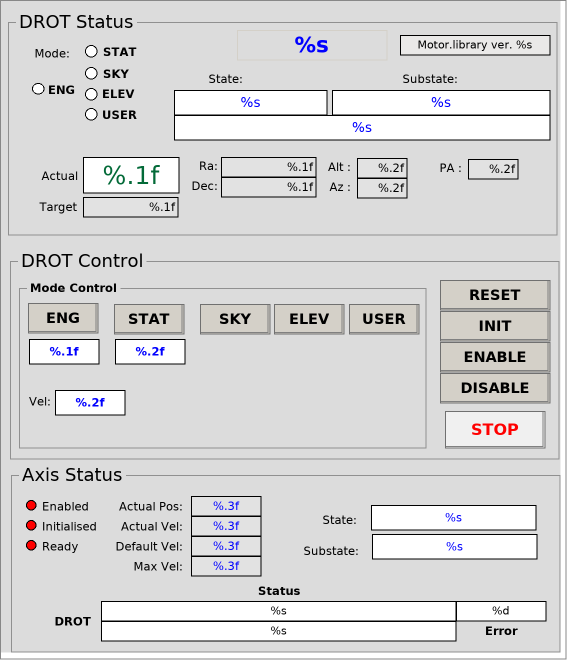
VISUALIZATION GUI_MA_DROT  // 567x660
    Frame (0,0 565x658)
        shows GUI_TEMPLATE_MA_DROT(m_DeviceName := 'DROT', m_Instance := MAIN.drot)
END_VISUALIZATION
